(* CODESYS project GustavoFonseca_RaonySantuzzi.project

Project tree, tasks and I/O mapping:
  Device : CODESYS Control Win V3, 3S - Smart Software Solutions GmbH, order no. 305021, version 3.5.11.40
    application Application
      libraries: Standard, * (System)
      task MainTask (cyclic, interval t#20ms, priority 1) calls PLC_PRG
      task Abastece (cyclic, interval 20 ms, priority 1) calls Tipo_De_Combustivel
      task Controla_Silos (cyclic, interval t#20ms, priority 1) calls Controla_Silos
      program PLC_PRG [ST]
      global variables GVL
      program ATUA_SCADA [ST]
      program ALARMES_SCADA [ST]
      program Tipo_De_Combustivel [ST]
      Types/
        data type COMBUSTIVEL
      program Controla_Silos [ST]
      program Reabastece_silos [ST]
*)

// Device/Application/Types/COMBUSTIVEL
{attribute 'qualified_only'}
{attribute 'strict'}
TYPE 
	COMBUSTIVEL : (ETANOL, GASOLINA_C, GASOLINA_P, NENHUM);
END_TYPE

// Device/Application/GVL
// Variáveis de Entrada (Sensores)
VAR_GLOBAL
	LIGA_AUTOMATICO : BOOL := FALSE ; (*comando de liga em moto automatico dado pelo supervisorio*)
	TIPO_COMBUSTIVEL : COMBUSTIVEL;
	
    LSH_S01 : BOOL := TRUE; (* Indicador de nível alto no silo S01 (>= 90%) *)
    LSH_S02 : BOOL := TRUE; (* Indicador de nível alto no silo S02 (>= 90%) *)
    LSH_S03 : BOOL := TRUE; (* Indicador de nível alto no silo S03 (>= 90%) *)
    LSL_S01 : BOOL := FALSE; (* Indicador de nível baixo no silo S01 (< 10%) *)
    LSL_S02 : BOOL := FALSE; (* Indicador de nível baixo no silo S02 (< 10%) *)
    LSL_S03 : BOOL := FALSE; (* Indicador de nível baixo no silo S03 (< 10%) *)
    LT_S01 : REAL := 100;  (* Transmissor ultrassônico indicando o nível do silo S01 (0-100%) *)
    LT_S02 : REAL := 100;  (* Transmissor ultrassônico indicando o nível do silo S02 (0-100%) *)
    LT_S03 : REAL := 100;  (* Transmissor ultrassônico indicando o nível do silo S03 (0-100%) *)
    Y_M_D1 : BOOL := FALSE;  (* Sensor de acoplamento da mangueira na doca 1 *)
    Y_M_D2 : BOOL := FALSE;  (* Sensor de acoplamento da mangueira na doca 2 *)
    Y_C_D1 : BOOL := FALSE;  (* Sensor de presença de caminhão na doca 1 *)
    Y_C_D2 : BOOL := FALSE;  (* Sensor de presença de caminhão na doca 2 *)
    EMERGENCIA : BOOL; (* Botão de emergência não retentivo *)
	ATIVA_EMERGENCIA : R_TRIG; (*Inicia o estado de emergência a partir da borda de subida do acionamento do botão de emergência*)
	REARME : BOOL; (* Botão de rearme não retentivo *)
	ATIVA_REARME : R_TRIG; (*Rearma o sistema a partir da borda de subida do acionamento do botão de rearme*)
	
    VA_S01 : BOOL := FALSE; (* Válvula de admissão do silo S01 *)
    VA_S02 : BOOL := FALSE; (* Válvula de admissão do silo S02 *)
    VA_S03 : BOOL := FALSE; (* Válvula de admissão do silo S03 *)
    VS_S01 : BOOL := FALSE; (* Válvula de escoamento do silo S01 *)
    VS_S02_1 : BOOL := FALSE; (* Válvula de escoamento do silo S02 para o tanque TQ1 *)
    VS_S02_2 : BOOL := FALSE; (* Válvula de escoamento do silo S02 para o tanque TQ2 *)
    VS_S03 : BOOL := FALSE; (* Válvula de escoamento do silo S03 *)
	VC_TQ1 : BOOL := FALSE; (*Valvula de liberação de combustivel na mangueira tanque 2*)
	VS_TQ2 : BOOL := FALSE; (*Valvula de liberação de combustivel na mangueira tanque 2*)
    M1 : BOOL := FALSE; (* Motor de agitação do tanque TQ1 *)
    M2 : BOOL := FALSE; (* Motor de agitação do tanque TQ2 *)
    B_R1 : BOOL := FALSE; (* Bomba de transporte do reservatório R1 para os silos S01 e S03 *)
    B_R2 : BOOL := FALSE; (* Bomba de transporte do reservatório R2 para o silo S02 *)
    C_D1 : BOOL := FALSE; (* Cancela de retenção da doca 1 *)
    C_D2 : BOOL := FALSE; (* Cancela de retenção da doca 2 *)
	
	BLOQ_ET : BOOL := FALSE;
	BLOQ_GAS_C : BOOL := FALSE;
	BLOQ_GAS_P : BOOL := FALSE;
	
    ABAST_AUTORIZADO : BOOL := FALSE;
	
	Caminhao_abastecido : BOOL := FALSE; 
	
	    // Alarmes relacionados aos níveis dos silos
    ALARME_NIVEL_ALTO_S01 : BOOL; (* Alarme de nível alto no silo S01 *)
    ALARME_NIVEL_BAIXO_S01 : BOOL; (* Alarme de nível baixo no silo S01 *)
    ALARME_NIVEL_ALTO_S02 : BOOL; (* Alarme de nível alto no silo S02 *)
    ALARME_NIVEL_BAIXO_S02 : BOOL; (* Alarme de nível baixo no silo S02 *)
    ALARME_NIVEL_ALTO_S03 : BOOL; (* Alarme de nível alto no silo S03 *)
    ALARME_NIVEL_BAIXO_S03 : BOOL; (* Alarme de nível baixo no silo S03 *)

    // Alarmes relacionados à desconexão incorreta de mangueiras
    ALARME_DESCONECT_MANGUEIRA_D1 : BOOL; (* Alarme de desconexão incorreta da mangueira na doca 1 *)
    ALARME_DESCONECT_MANGUEIRA_D2 : BOOL; (* Alarme de desconexão incorreta da mangueira na doca 2 *)

    // Alarme de emergência
    ALARME_EMERGENCIA : BOOL; (* Alarme de emergência acionado *)

    // Alarmes de operação
    ALARME_MISTURA_TQ1 : BOOL; (* Problema na mistura do tanque TQ1 *)
    ALARME_MISTURA_TQ2 : BOOL; (* Problema na mistura do tanque TQ2 *)

    // Alarmes gerais
    ALARME_OPERACAO_INVALIDA : BOOL; (* Operação inválida detectada *)

END_VAR

// Device/Application/PLC_PRG
PROGRAM PLC_PRG
VAR


END_VAR

IF GVL.LIGA_AUTOMATICO THEN
	IF GVL.Y_C_D1 AND GVL.Y_M_D1 THEN 
			GVL.C_D1 := TRUE; (*se o sensor de presença e o sensor de acoplamento da doca 1 estiverem OK, fecha a cancela doca1*)
	END_IF
	
	IF GVL.C_D1 THEN 
		IF GVL.TIPO_COMBUSTIVEL = COMBUSTIVEL.ETANOL AND NOT GVL.BLOQ_ET THEN (*Quando cancela fechada, aguandamos selecionar ETANOL*)
			GVL.BLOQ_GAS_C:= TRUE;
			GVL.BLOQ_GAS_P := TRUE;
			GVL.ABAST_AUTORIZADO := TRUE; (*Autoriza evento que dispara a tarefa Abastecimento*)
			//Tipo_Combustivel(TANQUE_CHEIO => Caminhao_abastecido ); (*Abre as valvulas e incrementa combustivel no caminhão até
                                                                      // que este esteja cheio, retorna caminhao abastecido*)		
		ELSIF GVL.TIPO_COMBUSTIVEL = COMBUSTIVEL.GASOLINA_C AND NOT GVL.BLOQ_GAS_C THEN
			GVL.BLOQ_ET:= TRUE;
			GVL.BLOQ_GAS_P := TRUE;
			GVL.ABAST_AUTORIZADO := TRUE;
			
		ELSIF GVL.TIPO_COMBUSTIVEL = COMBUSTIVEL.GASOLINA_P AND NOT GVL.BLOQ_GAS_P THEN
			GVL.BLOQ_ET := TRUE;
			GVL.BLOQ_GAS_C := TRUE;
			GVL.ABAST_AUTORIZADO := TRUE;
			
		END_IF
	END_IF
	
	IF GVL.Caminhao_abastecido THEN
		
		GVL.Caminhao_abastecido := FALSE;
		WHILE GVL.Y_M_D1 DO (*Aguarda que a mangueira seja desconectada*)
			IF GVL.Y_C_D1 THEN 
				GVL.ALARME_DESCONECT_MANGUEIRA_D1 := TRUE; (*Se detectado que o caminhao saiu antes de desconectar a mangueira
																	  um alarme de desconecta a mangueira é emitido*)
			END_IF
		END_WHILE
		
		GVL.C_D1 := FALSE; (*Cancela nao atuada, ou seja a cancela foi aberta*)
		(*Operacao finalizada*)

	END_IF
END_IF

END_PROGRAM

// Device/Application/Tipo_De_Combustivel
PROGRAM Tipo_De_Combustivel

VAR_OUTPUT
	TANQUE_CHEIO: BOOL := FALSE;
END_VAR

VAR
	
	Timer : TON;
	Tempo : REAL := 0 ; 
	Tempo_proporcao_etanol_GasC : REAL := 67;  (*  20ms * 67 = 1350 ms*) (*1350ms = 1,35s que corresponde ao tempo que S01 deve ficar aberta para a gasolina final
																	     ter uma porcentagem de 27%*)
	Tempo_proporcao_gasolina_GasC : REAL := 182;(*  20ms * 182 = 3650 ms*) (*3650ms = 3,65s que corresponde ao tempo que S02_1 deve ficar aberta para a gasolina final
																	     ter uma porcentagem de 27%*)
	
	NIVEL_CAMINHAO: REAL := 0; (*Indica o volume de combustivel carregado no caminhao*)
	
END_VAR


(*Se o combustivel selecionado for ETANOL:*)

IF GVL.TIPO_COMBUSTIVEL = COMBUSTIVEL.ETANOL THEN
GVL.VS_S01 := TRUE;
GVL.VC_TQ1 := TRUE;
Tempo := Tempo + 1;

IF Tempo <= 250 THEN (* 20ms * 250 = 5000 ms = 5 segundo, sendo uma vazao de 5000l/s e uma capacidade de 25000l do caminhao. 5 s é o tempo necessario para enche-lo*)
						
	NIVEL_CAMINHAO := NIVEL_CAMINHAO + 100;
	GVL.LT_S01 := GVL.LT_S01 - 0.002; (*Abaixa 0.002% no nivel do Silo 1, que equivale aos 100 l a cada 20ms*)

END_IF

END_IF

IF NIVEL_CAMINHAO >= 25000 THEN
	
	Tempo := 0;
	
	GVL.Caminhao_abastecido := TRUE; (*Sinaliza que o tanque do caminhao está cheio*)
	GVL.VS_S01 := FALSE;  
	GVL.VC_TQ1 := FALSE; (*Fecha as valvulas que liberam combustivel do tanque 1 para a mangueira*)
	
	GVL.BLOQ_GAS_C := FALSE; (*Desbloqueia os outros combustiveis para que eles possam ser solicitados*)
	GVL.BLOQ_GAS_P := FALSE;
	
	GVL.TIPO_COMBUSTIVEL := COMBUSTIVEL.NENHUM; 
	
END_IF


(* ////////// ///////// /////////*)



(*Se o combustivel selecionado for GASOLINA_C:*)

IF GVL.TIPO_COMBUSTIVEL = COMBUSTIVEL.GASOLINA_C THEN

GVL.VS_S02_1 := TRUE; 
GVL.VS_S01 := TRUE;
GVL.VC_TQ1 := TRUE;
Tempo := Tempo + 1;

IF Tempo < 67 THEN
	NIVEL_CAMINHAO := NIVEL_CAMINHAO + 100;
	GVL.LT_S01 := GVL.LT_S01 - 0.002; (*Abaixa 0.002% no nivel do Silo 1, que equivale aos 100 l a cada 20ms*) 
END_IF
IF Tempo < 182 THEN
	NIVEL_CAMINHAO := NIVEL_CAMINHAO + 100;
	GVL.LT_S02 := GVL.LT_S02 - 0.002;
END_IF


END_IF

IF NIVEL_CAMINHAO >= 25000 THEN
	
	GVL.Caminhao_abastecido := TRUE; (*Sinaliza que o tanque do caminhao está cheio*)
	GVL.VS_S01 := FALSE;  
	GVL.VC_TQ1 := FALSE; (*Fecha as valvulas que liberam combustivel do tanque 1 para a mangueira*)
	GVL.VS_S02_1 := FALSE;
	
	GVL.BLOQ_ET := FALSE; (*Desbloqueia os outros combustiveis para que eles possam ser solicitados*)
	GVL.BLOQ_GAS_P := FALSE;
	
	Tempo := 0;
	
	GVL.TIPO_COMBUSTIVEL := COMBUSTIVEL.NENHUM; 
	
END_IF

(* ////////// ///////// /////////*)




(*Se o combustivel selecionado for GASOLINA_P:*)

(* ////////// ///////// /////////*)

END_PROGRAM

// Device/Application/Controla_Silos
PROGRAM Controla_Silos (*Loop que fica constantemente checando se algum dos silos precisa ser reabastecido*)


VAR
	Enchendo_tanque :BOOL := FALSE; (*É uma variavel de realimentacao que mantem enchendo o 
									  tanque até q este chegue a capacidade maxima*)
END_VAR



IF GVL.LSL_S01 OR Enchendo_tanque THEN 
	GVL.VA_S01 := TRUE;
	GVL.B_R1 := TRUE;
	Enchendo_tanque := TRUE;
	
	IF (GVL.LT_S01 + 20) < 100 THEN
		GVL.LT_S01 := GVL.LT_S01 + 20;
	ELSE
		GVL.VA_S01 := FALSE;
		GVL.B_R1 := FALSE;
		Enchendo_tanque := FALSE;
	END_IF

END_IF

IF GVL.LT_S01 < 15 THEN (*Se o nivel estiver abaixo de 15 liga o indicador de nivel baixo *)
	GVL.LSL_S01 := TRUE;
	GVL.ALARME_NIVEL_BAIXO_S01 := TRUE;
ELSE
	GVL.LSL_S01 := FALSE;
	GVL.ALARME_NIVEL_BAIXO_S01 := FALSE;
END_IF 

IF GVL.LT_S01 > 95 THEN (*Se o nivel estiver acima de 95 liga o indicador de nival alto*)
	GVL.LSH_S01 := TRUE;
	GVL.ALARME_NIVEL_ALTO_S01 := TRUE;
ELSE
	GVL.LSH_S01 := FALSE;
	GVL.ALARME_NIVEL_ALTO_S01 := FALSE;

END_IF

END_PROGRAM

// Device/Application/ATUA_SCADA
PROGRAM ATUA_SCADA
VAR
	    // Variáveis de Interface para Entrada (Simuladas pelo SCADA)
		//INFORMAÇÕES ENVIADOS DO SCADA
    EMERGENCIA : BOOL; (* Botão de emergência retentivo *)
	
END_VAR

END_PROGRAM

// Device/Application/ALARMES_SCADA
PROGRAM ALARMES_SCADA
VAR
	

END_VAR

IF GVL.LSH_S01 THEN 
	GVL.ALARME_NIVEL_ALTO_S01 := TRUE; (*Emite alarme de nivel Alto em S01*)
ELSIF GVL.LSL_S01 THEN
	GVL.ALARME_NIVEL_BAIXO_S01 := TRUE; (*Emite alarme de nivel Baixo em S01*)
END_IF

IF GVL.LSH_S02 THEN 
	GVL.ALARME_NIVEL_ALTO_S02 := TRUE;
ELSIF GVL.LSL_S02 THEN
	GVL.ALARME_NIVEL_BAIXO_S02 := TRUE;
END_IF

IF GVL.LSH_S03 THEN 
	GVL.ALARME_NIVEL_ALTO_S03 := TRUE;
ELSIF GVL.LSL_S03 THEN
	GVL.ALARME_NIVEL_BAIXO_S03 := TRUE;
END_IF

END_PROGRAM

// Device/Application/Reabastece_silos
PROGRAM Reabastece_silos

VAR_INPUT
	SILO : REAL;
END_VAR

VAR
END_VAR


(*simula a abastecimento  do silo 1*)

IF GVL.LT_S01 <= 50 AND SILO = 1 THEN (*sE S01 estiver com o nivel abaixo de 50% ou seja, menos q o suficiente para encher um caminhao de etanol
						   por garantia ele sera reabastecido até 100% da capacidade*)
	GVL.VA_S01 := TRUE;
	GVL.B_R1 := TRUE;
	
	GVL.LT_S01 := GVL.LT_S01 + 20; (*A vazao de entrada é de 10000l o q equivale a um acrescimo de 20% por segundo *)
	
END_IF

(*simula a abastecimento do silo 2*)


IF GVL.LT_S02 <= 50 AND SILO = 2 THEN 
	
	GVL.VA_S02 := TRUE;
	GVL.B_R2 := TRUE;
	
	GVL.LT_S02 := GVL.LT_S02 + 20; 
	
END_IF

(*simula a abastecimento do silo 3*)

IF GVL.LT_S03 <= 50 AND SILO = 3 THEN 
	
	GVL.VA_S03 := TRUE;
	GVL.B_R1 := TRUE;
	
	GVL.LT_S03 := GVL.LT_S03 + 20; 
	
END_IF

END_PROGRAM
